PROGRAM PostNL
VAR
	Stap : INT;
	Timer: TON;
END_VAR


CASE stap OF
	
	0:	//Stap 0: Wachten op pakket van webshop
	IF GVL.TEMP_Overhandigen THEN
		stap := 1;
	END_IF
	
	
	
	1:	//Stap 1: Pakket binnen bij PostNL, wachten op sorteren
	IF GVL.BT_PakketSorteren THEN
		IF GVL.TEMP_OhpOfBezonrgen = TRUE THEN
			stap := 2;
			ELSIF GVL.TEMP_OhpOfBezonrgen = FALSE THEN
				stap := 3;
		END_IF
	END_IF
	
	
	
	2:	//Stap 2: Pakket ligt bij het ophaalpunt
	GVL.LED_PakketBijOHP := TRUE;
		
		//Wanneer pakket wordt opgehaald gaat het programma naar stap 3
		IF GVL.BT_BestellingOphalen THEN
			stap := 4;
		END_IF		
		
		
	
	3:
	//Start timer. Wanneer de deur na 10 seconden nog niet open is zal het pakket naar het ophaalpunt worden gebracht
	Timer(IN := TRUE, PT := T#10S);
		
	//Wacht tot deur open gaat
	IF GVL.BT_DeurOpen THEN
		Timer(IN := FALSE);
		stap := 4;
			
	//Gaat de deur niet open wordt het pakken naar het ophaalpunt gebracht (stap 4)
	ELSIF Timer.Q THEN
		Timer(IN := FALSE);
		stap := 2;
	END_IF
		
		
		
	4:	//Pakket is bezorgd
	GVL.LED_BestellingGeleverd := TRUE;
	GVL.LED_PakketBijOHP := FALSE;
		
END_CASE




//Aanroepen functie voor het tonen van de status van het pakket
IF GVL.BT_ToonStatus THEN
	GVL.TX_PakketInfo := TrackAndTraceInfo(stap);
END_IF

//Reset het programma naar stap 0
IF GVL.Reset THEN
	stap := 0;
END_IF

END_PROGRAM

(* stored: Version 1.1.0.1, ProductVersion 3.1.4024.13
   POU PostNL: Id {93e07b44-ce98-4bf0-8ee4-9a497784c1d4}, SpecialFunc None *)
